FUNCTION_BLOCK FB_Visitor IMPLEMENTS I_Visitor
VAR_INPUT
END_VAR
VAR_OUTPUT
END_VAR
VAR
END_VAR

METHOD VisitElementA
VAR_INPUT
	in_fbElementA	: FB_ElementA;
END_VAR
ADSLOGSTR(msgCtrlMask:= ADSLOG_MSGTYPE_ERROR, msgFmtStr:= 'I visit Element A right now', strArg:= '');
END_METHOD

{warning 'Add method implementation '}
METHOD VisitElementB
VAR_INPUT
	in_fbElementB	: FB_ElementB;
END_VAR
ADSLOGSTR(msgCtrlMask:= ADSLOG_MSGTYPE_ERROR, msgFmtStr:= 'I visit Element B right now', strArg:= '');
END_METHOD

END_FUNCTION_BLOCK

(* stored: Version 1.1.0.1
   POU FB_Visitor: Id {cb0b97f1-f59f-4311-9b9f-a2e71b83fde3}, SpecialFunc None
   Method VisitElementA: Id {b4c4afb0-bd14-4e88-88a3-24350b5a0e98}
   Method VisitElementB: Id {4611f983-5e3e-4451-8e1f-ea3040e336f1} *)
